FUNCTION F_ComputeFloatSize : UDINT
VAR_INPUT
    {attribute 'analysis' := '-33' }
    fValue : REAL;
END_VAR


F_ComputeFloatSize := GCL_PB.cFloatSize;

END_FUNCTION

(* stored: Version 1.1.0.1
   POU F_ComputeFloatSize: Id {a1759402-98e2-4ebb-be15-bdbbb9451038}, SpecialFunc None *)
